// TIA Portal V19 export
ORGANIZATION_BLOCK "Main"   // OB1, LAD, ProgramCycle
TITLE = "Main Program Sweep (Cycle)"
   VAR_TEMP
      OB1_EV_CLASS : Byte;   // Bits 0-3 = 1 (Coming event), Bits 4-7 = 1 (Event class 1)
      OB1_SCAN_1 : Byte;   // 1 (Cold restart scan 1 of OB 1), 3 (Scan 2-n of OB 1)
      OB1_PRIORITY : Byte;   // Priority of OB Execution
      OB1_OB_NUMBR : Byte;   // 1 (Organization block 1, OB1)
      OB1_RESERVED_1 : Byte;   // Reserved for system
      OB1_RESERVED_2 : Byte;   // Reserved for system
      OB1_PREV_CYCLE : Int;   // Cycle time of previous OB1 scan (milliseconds)
      OB1_MIN_CYCLE : Int;   // Minimum cycle time of OB1 (milliseconds)
      OB1_MAX_CYCLE : Int;   // Maximum cycle time of OB1 (milliseconds)
      OB1_DATE_TIME : Date_And_Time;   // Date and time OB1 started
   END_VAR
BEGIN

REGION Network 1
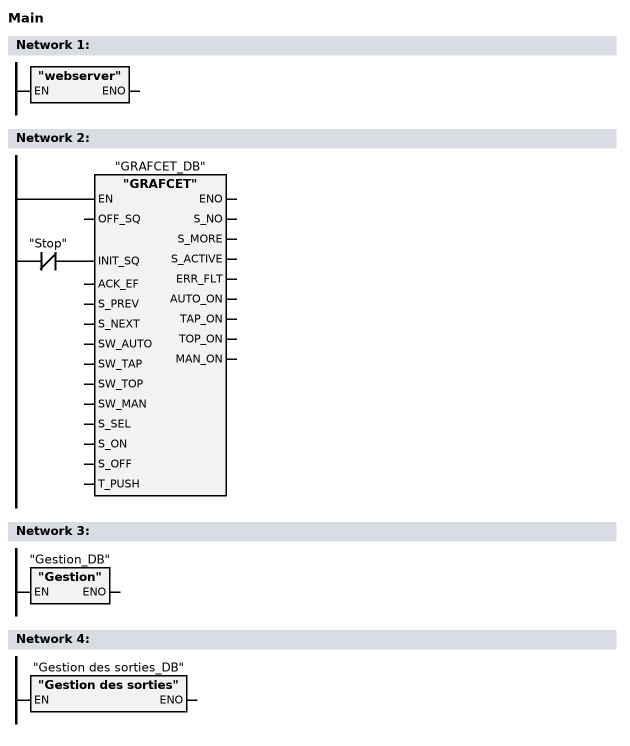
   RUNG wire#powerrail
      "webserver"()
   END_RUNG
   // the same network as SCL:
   "webserver"();
END_REGION

REGION Network 2
   RUNG wire#powerrail
      "GRAFCET_DB"(INIT_SQ := wire#w1, OFF_SQ :=, ACK_EF :=, S_PREV :=, S_NEXT :=, SW_AUTO :=, SW_TAP :=, SW_TOP :=, SW_MAN :=, S_SEL :=, S_ON :=, S_OFF :=, T_PUSH :=, S_NO =>, S_MORE =>, S_ACTIVE =>, ERR_FLT =>, AUTO_ON =>, TAP_ON =>, TOP_ON =>, MAN_ON =>)
   END_RUNG
   RUNG wire#powerrail
      I_Contact( "Stop" )
   END_RUNG wire#w1
   // the same network as SCL:
   "GRAFCET_DB"(INIT_SQ := NOT "Stop");   // "GRAFCET"
END_REGION

REGION Network 3
   RUNG wire#powerrail
      "Gestion_DB"()
   END_RUNG
   // the same network as SCL:
   "Gestion_DB"();   // "Gestion"
END_REGION

REGION Network 4
   RUNG wire#powerrail
      "Gestion des sorties_DB"()
   END_RUNG
   // the same network as SCL:
   "Gestion des sorties_DB"();   // "Gestion des sorties"
END_REGION

NETWORK
TITLE = Call system diagnostics block
      CALL  "RSE_FB", "RSE_DB";
END_ORGANIZATION_BLOCK
